PROGRAM MAIN
VAR
	test : EventLoggerClass;
END_VAR

test();

END_PROGRAM

(* stored: Version 1.1.0.1, ProductVersion 3.1.4024.9
   POU MAIN: Id {902d5820-3fe0-4aff-8c96-1938b68e5f95}, SpecialFunc None *)
